// TIA Portal V18 export
FUNCTION_BLOCK "defects_util"   // FB31, FBD
{ S7_Optimized_Access := 'TRUE' }
VERSION : 0.1
// stored: AutoNumber true, IsIECCheckEnabled false, IsRetainMemResEnabled false, MemoryReserve 100, SetENOAutomatically false, UDAEnableTagReadback false
   VAR_INPUT
      ALLOWED : Bool;
      xBdefect_inc : Bool;
      xBdefect_dec : Bool;
      xDefectsClearAll : Bool;
      xDefect_Save : Bool;
      positions : "typePositions";
   END_VAR
   VAR_OUTPUT
      go_to_defect_now : Bool;
   END_VAR
   VAR_IN_OUT
      xyBeepDone : Bool;
      DEFECTS_DB : "typeDefectsDB";
   END_VAR
   VAR
      mem1 : Bool;
      mem2 : Bool;
      xdefect_dec_was : Bool;
      xdefect_inc_was : Bool;
      xDefect_Save_was : Bool;
      xDefectsClearAll_was : Bool;
   END_VAR
BEGIN

REGION Network 1 (SCL)
   IF #ALLOWED THEN
       IF #xBdefect_inc AND NOT #xdefect_inc_was THEN
           IF #DEFECTS_DB.N >0 THEN
               IF #DEFECTS_DB.i < #DEFECTS_DB.N THEN
                   #DEFECTS_DB.i := #DEFECTS_DB.i + 1;
                   #go_to_defect_now := true;
               ELSE
                   #xyBeepDone := true;
                   #DEFECTS_DB.i := #DEFECTS_DB.N;
               END_IF;
               #xyBeepDone := true;
           END_IF;
       END_IF;


       IF #xBdefect_dec AND NOT #xdefect_dec_was THEN
           IF #DEFECTS_DB.i > 1 THEN
               #DEFECTS_DB.i := #DEFECTS_DB.i - 1;
               #go_to_defect_now := true;
           ELSE
               #DEFECTS_DB.i :=  1;
               #xyBeepDone := true;
           END_IF;
       END_IF;
       IF NOT #xBdefect_inc AND NOT #xBdefect_dec THEN
           #go_to_defect_now := false;
       END_IF;

   ELSE
       #go_to_defect_now := false;
   END_IF;


   #xdefect_inc_was := #xBdefect_inc;
   #xdefect_dec_was := #xBdefect_dec;
END_REGION

REGION Network 2 (SCL)
   IF #xDefect_Save AND NOT #xDefect_Save_was THEN
       IF #DEFECTS_DB.N < #DEFECTS_DB.N_max THEN
           #DEFECTS_DB.pos_AR[#DEFECTS_DB.N] := "_MAIN_DB".Mot_Positions;
           #DEFECTS_DB.N := #DEFECTS_DB.N + 1;
       ELSE
           #xyBeepDone := true;
       END_IF;
   END_IF;

   #xDefect_Save_was := #xDefect_Save;


   IF #xDefectsClearAll AND NOT #xDefectsClearAll_was THEN
       #DEFECTS_DB.N := 0;
       #DEFECTS_DB.i := 0;

   END_IF;
   #xDefectsClearAll_was := #xDefectsClearAll;
END_REGION
END_FUNCTION_BLOCK
